VAR_GLOBAL
END_VAR

(* stored: Version 1.1.0.1, ProductVersion 3.1.0.26
   GVL GVL: Id {e5bd4bfe-337e-49ca-b9b9-232e4d92833a} *)
